// TIA Portal V20 export
// export: Created 2025-12-01T14:56:13.507243Z, ExportSetting None, DisplayName Totally Integrated Automation Portal, DisplayVersion V20 Update 3, DisplayName TIA Portal Openness, DisplayVersion V20 Update 3, DisplayName TIA Portal Version Control Interface, DisplayVersion V20 Update 3, DisplayName STEP 7 Professional, DisplayVersion V20 Update 3, DisplayName STEP 7 Safety, DisplayVersion V20 Update 2, DisplayName WinCC Basic/Comfort/Advanced, DisplayVersion V20 Update 3, DisplayName WinCC Professional, DisplayVersion V20 Update 3, DisplayName WinCC Unified, DisplayVersion V20 Update 3
TYPE "UDT_ProtocoloEmiMesa"
   STRUCT
      PresRouter : Bool;
      PresNormal : Bool;   // Presencia Normal
      Ausencia : Bool;   // Ausencia
      PresBloqueo : Bool;   // Presencia Bloqueo
      PresGalibo : Bool;   // Presencia con Galibo
      Bit_05 : Bool;
      Bit_06 : Bool;
      PresReset : Bool;   // Presencia del Reset
      Bit_10 : Bool;
      Bit_11 : Bool;
      Bit_12 : Bool;
      Bit_13 : Bool;
      Bit_14 : Bool;
      Bit_15 : Bool;
      Bit_16 : Bool;
      RecepOK : Bool;   // Recepcion OK de la Orden
   END_STRUCT;
END_TYPE
